Staubli VAL3: link_it.pgx

public program link_it(string x_sName)
begin
  // link all the point
  call link_all(x_sName)
  // put the base config
  tTraj[x_sName].tData[0].tSuper.moveType=1
end
